{attribute 'qualified_only'}
VAR_GLOBAL
	//
END_VAR

(* stored: Version 1.1.0.1, ProductVersion 3.1.4024.12
   GVL GVL_IO: Id {5c43743a-db06-47f7-8502-86473cb3cb44} *)
